% RSLogix 500 project INVENTORY_CHECK_BAK043.RSS, saved by version 12.00.00.00 %
PROJECT "UNTITLED"    % processor: Bul.1763 MicroLogix 1100 Series B %

PROGRAM FILES
  LAD 2 "MAIN"  16 rungs

DATA FILES
  O0 OUTPUT  4 elements
  I1 INPUT  6 elements
  S2 STATUS  66 elements
  B3 BINARY  1 elements
  T4 TIMER  1 elements
  C5 COUNTER  1 elements
  R6 CONTROL  1 elements
  N7 INTEGER  11 elements
  F8 FLOAT  1 elements
  ST9 STRING  7 elements

LADDER 2 "MAIN"
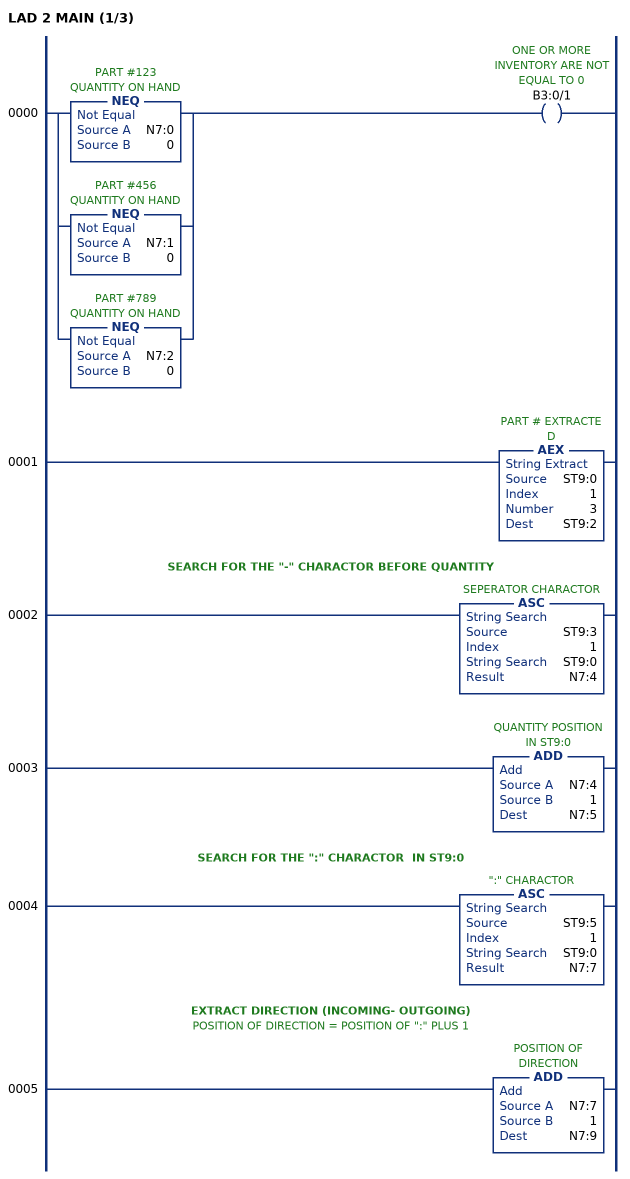
% Rung: 0 %
SOR BST NEQ N7:0 0 NXB NEQ N7:1 0 NXB NEQ N7:2 0 BND OTE B3:0/1 EOR
%   N7:0  "PART #123 QUANTITY ON HAND" %
%   N7:1  "PART #456 QUANTITY ON HAND" %
%   N7:2  "PART #789 QUANTITY ON HAND" %
%   B3:0/1  "ONE OR MORE INVENTORY ARE NOT EQUAL TO 0" %
% Rung: 1 %
SOR AEX ST9:0 1 3 ST9:2 EOR
%   ST9:0  "BARCODE SCAN TO PLC" %
%   ST9:2  "PART # EXTRACTED" %
% Rung: 2 %
% TITLE: SEARCH FOR THE "-" CHARACTOR BEFORE QUANTITY %
SOR ASC ST9:3 1 ST9:0 N7:4 EOR
%   ST9:3  "SEPERATOR CHARACTOR" %
%   ST9:0  "BARCODE SCAN TO PLC" %
%   N7:4  "SEPERATOR POSITION" %
% Rung: 3 %
SOR ADD N7:4 1 N7:5 EOR
%   N7:4  "SEPERATOR POSITION" %
%   N7:5  "QUANTITY POSITION IN ST9:0" %
% Rung: 4 %
% TITLE: SEARCH FOR THE ":" CHARACTOR  IN ST9:0 %
SOR ASC ST9:5 1 ST9:0 N7:7 EOR
%   ST9:5  "":" CHARACTOR" %
%   ST9:0  "BARCODE SCAN TO PLC" %
%   N7:7  "POSITION OF ":"" %
% Rung: 5 %
% TITLE: EXTRACT DIRECTION (INCOMING- OUTGOING) %
% POSITION OF DIRECTION = POSITION OF ":" PLUS 1 %
SOR ADD N7:7 1 N7:9 EOR
%   N7:7  "POSITION OF ":"" %
%   N7:9  "POSITION OF DIRECTION" %

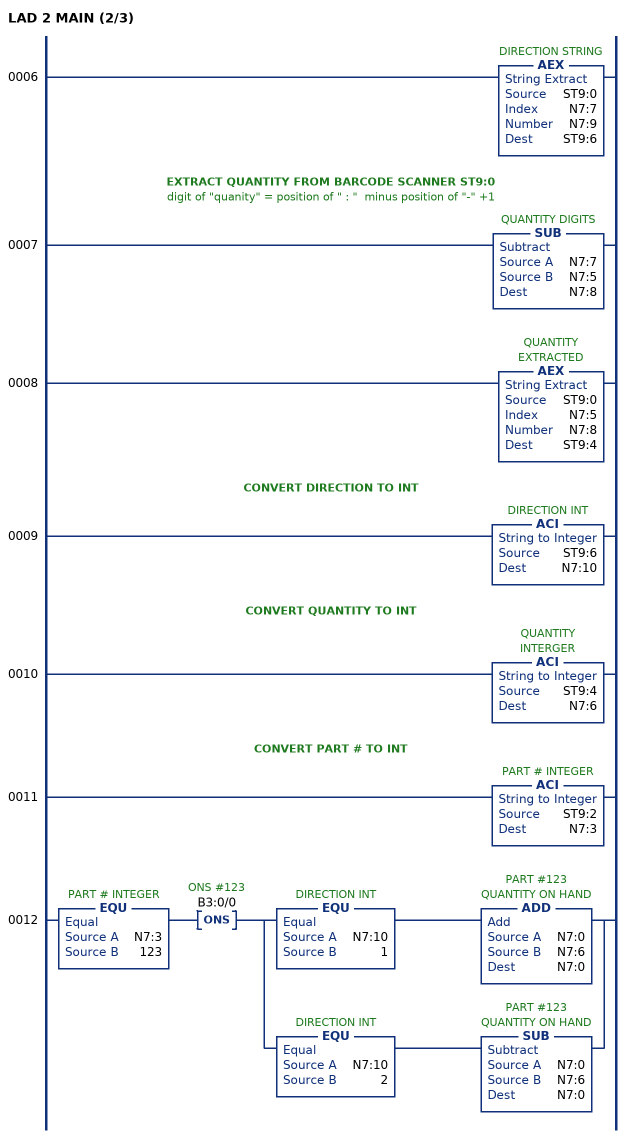
% Rung: 6 %
SOR AEX ST9:0 N7:7 N7:9 ST9:6 EOR
%   ST9:0  "BARCODE SCAN TO PLC" %
%   N7:7  "POSITION OF ":"" %
%   N7:9  "POSITION OF DIRECTION" %
%   ST9:6  "DIRECTION STRING" %
% Rung: 7 %
% TITLE: EXTRACT QUANTITY FROM BARCODE SCANNER ST9:0 %
% digit of "quanity" = position of " : "  minus position of "-" +1 %
SOR SUB N7:7 N7:5 N7:8 EOR
%   N7:7  "POSITION OF ":"" %
%   N7:5  "QUANTITY POSITION IN ST9:0" %
%   N7:8  "QUANTITY DIGITS" %
% Rung: 8 %
SOR AEX ST9:0 N7:5 N7:8 ST9:4 EOR
%   ST9:0  "BARCODE SCAN TO PLC" %
%   N7:5  "QUANTITY POSITION IN ST9:0" %
%   N7:8  "QUANTITY DIGITS" %
%   ST9:4  "QUANTITY EXTRACTED" %
% Rung: 9 %
% TITLE: CONVERT DIRECTION TO INT %
SOR ACI ST9:6 N7:10 EOR
%   ST9:6  "DIRECTION STRING" %
%   N7:10  "DIRECTION INT" %
% Rung: 10 %
% TITLE: CONVERT QUANTITY TO INT %
SOR ACI ST9:4 N7:6 EOR
%   ST9:4  "QUANTITY EXTRACTED" %
%   N7:6  "QUANTITY INTERGER" %
% Rung: 11 %
% TITLE: CONVERT PART # TO INT %
SOR ACI ST9:2 N7:3 EOR
%   ST9:2  "PART # EXTRACTED" %
%   N7:3  "PART # INTEGER" %
% Rung: 12 %
SOR EQU N7:3 123 ONS B3:0/0 BST EQU N7:10 1 ADD N7:0 N7:6 N7:0 NXB EQU N7:10 2 SUB N7:0 N7:6 N7:0 BND EOR
%   N7:3  "PART # INTEGER" %
%   B3:0/0  "ONS #123" %
%   N7:10  "DIRECTION INT" %
%   N7:0  "PART #123 QUANTITY ON HAND" %
%   N7:6  "QUANTITY INTERGER" %

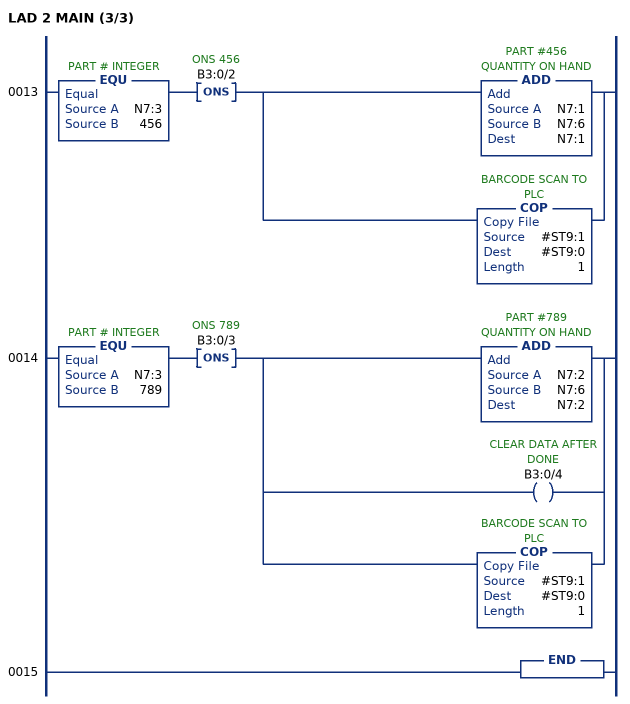
% Rung: 13 %
SOR EQU N7:3 456 ONS B3:0/2 BST ADD N7:1 N7:6 N7:1 NXB COP #ST9:1 #ST9:0 1 BND EOR
%   N7:3  "PART # INTEGER" %
%   B3:0/2  "ONS 456" %
%   N7:1  "PART #456 QUANTITY ON HAND" %
%   N7:6  "QUANTITY INTERGER" %
%   ST9:1  "RESET TO 0" %
%   ST9:0  "BARCODE SCAN TO PLC" %
% Rung: 14 %
SOR EQU N7:3 789 ONS B3:0/3 BST ADD N7:2 N7:6 N7:2 NXB OTE B3:0/4 NXB COP #ST9:1 #ST9:0 1 BND EOR
%   N7:3  "PART # INTEGER" %
%   B3:0/3  "ONS 789" %
%   N7:2  "PART #789 QUANTITY ON HAND" %
%   N7:6  "QUANTITY INTERGER" %
%   B3:0/4  "CLEAR DATA AFTER DONE" %
%   ST9:1  "RESET TO 0" %
%   ST9:0  "BARCODE SCAN TO PLC" %
% Rung: 15 %
SOR END EOR

OTHER DOCUMENTED ADDRESSES
  B3:0/5  "INPUT TO INVENTORY"

DATA TABLE (non-zero values as saved)
DATA ST9
% ST9:1 % "0"
% ST9:3 % "-"
% ST9:5 % ":"
